TYPE ST_StepBranch_1 :
STRUCT    
    NextStep        : DINT;
    Condition       : ARRAY [1..16] OF BOOL;
    ConditionMet    : BOOL;
END_STRUCT
END_TYPE

(* stored: Version 1.1.0.1, ProductVersion 3.1.4024.12
   DUT ST_StepBranch_1: Id {359e8df5-b3dd-4950-9a7a-9857f95267ad} *)
